FUNCTION_BLOCK PUBLIC ACMethodExtruding EXTENDS ACMethodRouteBase
VAR_INPUT
END_VAR
VAR_OUTPUT
END_VAR
VAR
END_VAR
VAR PERSISTENT
	_Parameter : ACMethodExtrudingP;
	_Result : ACMethodExtrudingR;
END_VAR

PROPERTY IsValid : BOOL
GET
IsValid := TRUE;
END_GET
END_PROPERTY

PROPERTY Parameter : ACMethodExtrudingP
GET
Parameter := _Parameter;
END_GET
SET
_Parameter := Parameter;
END_SET
END_PROPERTY

PROPERTY Result : ACMethodExtrudingR
GET
Result := _Result;
END_GET
SET
_Result := Result;
END_SET
END_PROPERTY

END_FUNCTION_BLOCK

(* stored: Version 1.1.0.1, ProductVersion 3.1.4020.12
   POU ACMethodExtruding: Id {2810847e-45bc-44fd-94c1-f87f3f71e814}, SpecialFunc None
   Property IsValid: Id {aa182da7-8a9b-4a00-9d81-2775e6857682}
   Get Get: Id {038c9ca3-35bf-47b8-a0a7-fc4dc421fa97}
   Property Parameter: Id {7952bdf4-4c46-4638-9234-93596d89c927}
   Get Get: Id {7322d8bf-9374-4083-b4c2-0384e004394d}
   Set Set: Id {6ab06d95-34c2-47d7-8e56-ce589c7b7d1a}
   Property Result: Id {0b346fe3-01ae-432b-9ac9-d4a44bd9ab5d}
   Get Get: Id {22594cc4-7b8a-47b6-af24-f219beb5fe4b}
   Set Set: Id {f59db4ab-9167-47e9-9301-445f446be1ff} *)
